{attribute addProperty BoxType "AX8620-1000-0026"}
{attribute addProperty Id "StatuswordAT %I*Statusword_3B58AC51162"}
{attribute addProperty CRC "854043290"}
{attribute addProperty SizeInBites "16"}
{attribute addProperty SizeInBytes "2"}
TYPE PSM_PSM_Statusword_32E7AA9A :
STRUCT
	{attribute addProperty Name "Statusword"}
	Statusword AT %I* : Statusword_3B58AC51;
END_STRUCT
END_TYPE

(* stored: Version 1.2.0.0, ProductVersion 3.1.4024.9
   DUT PSM_PSM_Statusword_32E7AA9A: Id {cb69a5ab-2d27-4c37-8fb1-31f1470c00c9} *)
